// TIA Portal V18 export
// export: Created 2026-01-09T11:32:05.3383076Z, ExportSetting WithDefaults, DisplayName Totally Integrated Automation Portal, DisplayVersion V18 Update 5, DisplayName TIA Portal Openness, DisplayVersion V18 Update 5, DisplayName TIA Portal Teamcenter Gateway, DisplayVersion V18, DisplayName TIA Portal Version Control Interface, DisplayVersion V18, DisplayName SINAMICS Startdrive Advanced, DisplayVersion V18 SP2 Update 1, DisplayName SINAMICS Startdrive G110M, G120, G120C, G120D, G120P, G115D, DisplayVersion V18 SP2 Update 1, DisplayName SINAMICS Startdrive G130, G150, S120, S150, SINAMICS MV, S210, G220, S200, DisplayVersion V18 SP2 Update 1, DisplayName STEP 7 Professional, DisplayVersion V18 Update 5, DisplayName STEP 7 Safety, DisplayVersion V18, DisplayName WinCC Professional, DisplayVersion V18 Update 5
TagTable "CyConfig"
  gloCyVisual_CyConfigCount{0,0} : Byte  (%DB[ST_CyDBNum].DBB136, CPU S71500-2PN_TP700, 1 s)
  gloCyVisual_CyConfigCount{0,1} : Byte  (%DB[ST_CyDBNum].DBB137, CPU S71500-2PN_TP700, 1 s)
  gloCyVisual_CyConfigCount{1,0} : Byte  (%DB[ST_CyDBNum].DBB138, CPU S71500-2PN_TP700, 1 s)
  gloCyVisual_CyConfigCount{1,1} : Byte  (%DB[ST_CyDBNum].DBB139, CPU S71500-2PN_TP700, 1 s)
  gloCyVisual_CyConfigCount{2,0} : Byte  (%DB[ST_CyDBNum].DBB140, CPU S71500-2PN_TP700, 1 s)
  gloCyVisual_CyConfigCount{2,1} : Byte  (%DB[ST_CyDBNum].DBB141, CPU S71500-2PN_TP700, 1 s)
  gloCyVisual_CyConfigCount{3,0} : Byte  (%DB[ST_CyDBNum].DBB142, CPU S71500-2PN_TP700, 1 s)
  gloCyVisual_CyConfigCount{3,1} : Byte  (%DB[ST_CyDBNum].DBB143, CPU S71500-2PN_TP700, 1 s)
  gloCyVisual_CyConfigCount{4,0} : Byte  (%DB[ST_CyDBNum].DBB144, CPU S71500-2PN_TP700, 1 s)
  gloCyVisual_CyConfigCount{4,1} : Byte  (%DB[ST_CyDBNum].DBB145, CPU S71500-2PN_TP700, 1 s)
  gloCyVisual_CyEnd : Byte  (%DB[ST_CyDBNum].DBB201, CPU S71500-2PN_TP700, 1 s)
  gloCyVisual_CyStart : Byte  (%DB[ST_CyDBNum].DBB200, CPU S71500-2PN_TP700, 1 s)
  gloCyVisual_CyConfigCount{5,0} : Byte  (%DB[ST_CyDBNum].DBB146, CPU S71500-2PN_TP700, 1 s)
  gloCyVisual_CyConfigCount{5,1} : Byte  (%DB[ST_CyDBNum].DBB147, CPU S71500-2PN_TP700, 1 s)
  gloCyVisual_CyConfigCount{6,0} : Byte  (%DB[ST_CyDBNum].DBB148, CPU S71500-2PN_TP700, 1 s)
  gloCyVisual_CyConfigCount{6,1} : Byte  (%DB[ST_CyDBNum].DBB149, CPU S71500-2PN_TP700, 1 s)
  gloCyVisual_CyConfigCount{7,0} : Byte  (%DB[ST_CyDBNum].DBB150, CPU S71500-2PN_TP700, 1 s)
  gloCyVisual_CyConfigCount{7,1} : Byte  (%DB[ST_CyDBNum].DBB151, CPU S71500-2PN_TP700, 1 s)
  gloCyVisual_CyConfigCount{8,0} : Byte  (%DB[ST_CyDBNum].DBB152, CPU S71500-2PN_TP700, 1 s)
  gloCyVisual_CyConfigCount{8,1} : Byte  (%DB[ST_CyDBNum].DBB153, CPU S71500-2PN_TP700, 1 s)
  gloCyVisual_CyConfigCount{9,0} : Byte  (%DB[ST_CyDBNum].DBB154, CPU S71500-2PN_TP700, 1 s)
  gloCyVisual_CyConfigCount{9,1} : Byte  (%DB[ST_CyDBNum].DBB155, CPU S71500-2PN_TP700, 1 s)
  gloCyVisual_CyConfigCount{10,0} : Byte  (%DB[ST_CyDBNum].DBB156, CPU S71500-2PN_TP700, 1 s)
  gloCyVisual_CyConfigCount{10,1} : Byte  (%DB[ST_CyDBNum].DBB157, CPU S71500-2PN_TP700, 1 s)
  gloCyVisual_CyConfigCount{11,0} : Byte  (%DB[ST_CyDBNum].DBB158, CPU S71500-2PN_TP700, 1 s)
  gloCyVisual_CyConfigCount{11,1} : Byte  (%DB[ST_CyDBNum].DBB159, CPU S71500-2PN_TP700, 1 s)
  gloCyVisual_CyConfigCount{12,0} : Byte  (%DB[ST_CyDBNum].DBB160, CPU S71500-2PN_TP700, 1 s)
  gloCyVisual_CyConfigCount{12,1} : Byte  (%DB[ST_CyDBNum].DBB161, CPU S71500-2PN_TP700, 1 s)
  gloCyVisual_CyConfigCount{13,0} : Byte  (%DB[ST_CyDBNum].DBB162, CPU S71500-2PN_TP700, 1 s)
  gloCyVisual_CyConfigCount{13,1} : Byte  (%DB[ST_CyDBNum].DBB163, CPU S71500-2PN_TP700, 1 s)
  gloCyVisual_CyConfigCount{14,0} : Byte  (%DB[ST_CyDBNum].DBB164, CPU S71500-2PN_TP700, 1 s)
  gloCyVisual_CyConfigCount{14,1} : Byte  (%DB[ST_CyDBNum].DBB165, CPU S71500-2PN_TP700, 1 s)
  gloCyVisual_CyConfigCount{15,0} : Byte  (%DB[ST_CyDBNum].DBB166, CPU S71500-2PN_TP700, 1 s)
  gloCyVisual_CyConfigCount{15,1} : Byte  (%DB[ST_CyDBNum].DBB167, CPU S71500-2PN_TP700, 1 s)
  gloCyVisual_CyConfigCount{16,0} : Byte  (%DB[ST_CyDBNum].DBB168, CPU S71500-2PN_TP700, 1 s)
  gloCyVisual_CyConfigCount{16,1} : Byte  (%DB[ST_CyDBNum].DBB169, CPU S71500-2PN_TP700, 1 s)
  gloCyVisual_CyConfigCount{17,0} : Byte  (%DB[ST_CyDBNum].DBB170, CPU S71500-2PN_TP700, 1 s)
  gloCyVisual_CyConfigCount{17,1} : Byte  (%DB[ST_CyDBNum].DBB171, CPU S71500-2PN_TP700, 1 s)
  gloCyVisual_CyConfigCount{18,0} : Byte  (%DB[ST_CyDBNum].DBB172, CPU S71500-2PN_TP700, 1 s)
  gloCyVisual_CyConfigCount{18,1} : Byte  (%DB[ST_CyDBNum].DBB173, CPU S71500-2PN_TP700, 1 s)
  gloCyVisual_CyConfigCount{19,0} : Byte  (%DB[ST_CyDBNum].DBB174, CPU S71500-2PN_TP700, 1 s)
  gloCyVisual_CyConfigCount{19,1} : Byte  (%DB[ST_CyDBNum].DBB175, CPU S71500-2PN_TP700, 1 s)
  gloCyVisual_CyConfigCount{20,0} : Byte  (%DB[ST_CyDBNum].DBB176, CPU S71500-2PN_TP700, 1 s)
  gloCyVisual_CyConfigCount{20,1} : Byte  (%DB[ST_CyDBNum].DBB177, CPU S71500-2PN_TP700, 1 s)
  gloCyVisual_CyConfigCount{21,0} : Byte  (%DB[ST_CyDBNum].DBB178, CPU S71500-2PN_TP700, 1 s)
  gloCyVisual_CyConfigCount{21,1} : Byte  (%DB[ST_CyDBNum].DBB179, CPU S71500-2PN_TP700, 1 s)
  gloCyVisual_CyConfigCount{22,0} : Byte  (%DB[ST_CyDBNum].DBB180, CPU S71500-2PN_TP700, 1 s)
  gloCyVisual_CyConfigCount{22,1} : Byte  (%DB[ST_CyDBNum].DBB181, CPU S71500-2PN_TP700, 1 s)
  gloCyVisual_CyConfigCount{23,0} : Byte  (%DB[ST_CyDBNum].DBB182, CPU S71500-2PN_TP700, 1 s)
  gloCyVisual_CyConfigCount{23,1} : Byte  (%DB[ST_CyDBNum].DBB183, CPU S71500-2PN_TP700, 1 s)
  gloCyVisual_CyConfigCount{24,0} : Byte  (%DB[ST_CyDBNum].DBB184, CPU S71500-2PN_TP700, 1 s)
  gloCyVisual_CyConfigCount{24,1} : Byte  (%DB[ST_CyDBNum].DBB185, CPU S71500-2PN_TP700, 1 s)
  gloCyVisual_CyConfigCount{25,0} : Byte  (%DB[ST_CyDBNum].DBB186, CPU S71500-2PN_TP700, 1 s)
  gloCyVisual_CyConfigCount{25,1} : Byte  (%DB[ST_CyDBNum].DBB187, CPU S71500-2PN_TP700, 1 s)
  gloCyVisual_CyConfigCount{26,0} : Byte  (%DB[ST_CyDBNum].DBB188, CPU S71500-2PN_TP700, 1 s)
  gloCyVisual_CyConfigCount{26,1} : Byte  (%DB[ST_CyDBNum].DBB189, CPU S71500-2PN_TP700, 1 s)
  gloCyVisual_CyConfigCount{27,0} : Byte  (%DB[ST_CyDBNum].DBB190, CPU S71500-2PN_TP700, 1 s)
  gloCyVisual_CyConfigCount{27,1} : Byte  (%DB[ST_CyDBNum].DBB191, CPU S71500-2PN_TP700, 1 s)
  gloCyVisual_CyConfigCount{28,0} : Byte  (%DB[ST_CyDBNum].DBB192, CPU S71500-2PN_TP700, 1 s)
  gloCyVisual_CyConfigCount{28,1} : Byte  (%DB[ST_CyDBNum].DBB193, CPU S71500-2PN_TP700, 1 s)
  gloCyVisual_CyConfigCount{29,0} : Byte  (%DB[ST_CyDBNum].DBB194, CPU S71500-2PN_TP700, 1 s)
  gloCyVisual_CyConfigCount{29,1} : Byte  (%DB[ST_CyDBNum].DBB195, CPU S71500-2PN_TP700, 1 s)
